PROGRAM demo3
VAR
	runner : FB_TaskRunner(ContainerType.PARALLEL_QUEUE);

	init: BOOL;
	_state :UINT;
	mc_power : FutureMCPower;
	_handl_power_on	: I_Job;
	_handl_demo_job : I_Job;
	
	_today : TIMESTRUCT;

	bPower : BOOL;
	bStart : BOOL;

	motion_data : ST_MotionData;	
	demo_job_container : FB_BatchJobContainer;
	i : UDINT;
END_VAR

IF NOT init THEN
	JobCreateDemo(demo_job_container, GVL.axis1); // demo_job にメソッドを通してシーケンスジョブを組み立てる
	mc_power.future_name := 'POWER_CTRL';
	init := TRUE;	// RUN 後 1 サイクルだけ実行
END_IF

_today := FILETIME64_TO_SYSTEMTIME(runner.current_time);
runner(root_job_name := 'ROOT',root_job_serial := (_today.wYear MOD 100) * 10000 + _today.wMonth * 100 + _today.wDay);

// Axis
GVL.axis1.ReadStatus();
MEMCPY(ADR(motion_data), ADR(GVL.axis1.NcToPlc), SIZEOF(GVL.axis1.NcToPlc));
motion_data.record_time := runner.current_time;

CASE _state OF
	0:
		IF bPower THEN
			mc_power.set_parameters(axis := GVL.axis1, status := TRUE); // Servo on
			_handl_power_on := runner.append_future(mc_power);
			_state := 1;
		END_IF
	1:
		IF _handl_power_on.ready THEN
			_handl_power_on.start();
		END_IF
		IF _handl_power_on.done THEN
			_state := 2;
		END_IF
	2:
		IF bStart THEN
			_handl_demo_job := runner.append_future(demo_job_container);
			_state := 3;
		END_IF
	3:
		IF _handl_demo_job.ready THEN
			_handl_demo_job.start();
		END_IF
		IF _handl_demo_job.current_state = E_FutureExecutionState.finish THEN
			_state := 2;
			//bStart := FALSE;
		END_IF
		IF NOT bPower THEN
			_state := 4;
		END_IF
	4:
		IF runner.halt(_handl_demo_job) THEN
			_state := 5;
		END_IF
	5:
		mc_power.set_parameters(axis := GVL.axis1, status := FALSE); // Servo off
		_handl_power_on := runner.append_future(mc_power);
		_state := 6;
	6:
		IF _handl_power_on.ready THEN
			_handl_power_on.start();
		END_IF
		IF _handl_power_on.done THEN
			_state := 0;
		END_IF
END_CASE

//IF _state > 0 AND NOT bPower THEN
//END_IF

METHOD JobCreateDemo : BOOL
VAR_INPUT
	job_container : I_Container;
	stAxis1	: REFERENCE TO AXIS_REF;
END_VAR
VAR
	_base_future : I_Future;
	_job_temp : I_Job;
	_job_temp_parent : I_Job;
	sleep : POINTER TO FutureSleep;
	sleep_creator : FutureSleepCreator;

	//mc_move_rel_future : POINTER TO FutureMCMoveRelative;
	mc_move_rel_future_creator : FutureMCMoveRelativeCreator;

	//mc_move_abs_future : POINTER TO FutureMCMoveAbsolute;
	mc_move_abs_future_creator : FutureMCMoveAbsoluteCreator;

	//mc_move_velocity_future: POINTER TO FutureMCMoveVelocity;
	mc_move_velocity_future_creator: FutureMCMoveVelocityCreator;
	
	mc_stop_future_creator : FutureMcStopCreator;
	
	i : UDINT;

END_VAR
//base_job.create_container(ContainerTYpe.BATCH, 'DEMO_JOB');
IF __QUERYINTERFACE(job_container,_base_future) THEN
	_base_future.future_name := 'JOB ROOT';
END_IF

// Sequence
_job_temp_parent := job_container.create_container(ContainerTYpe.BATCH, 'STEP MOVING');
FOR i := 1 TO 4 DO

	mc_move_rel_future_creator.set_parameters(stAxis1,20,200,0,0,0,0);
	_job_temp := _job_temp_parent.children.create_job(mc_move_rel_future_creator,'Move +20 deg, 200 deg/s');

	sleep_creator.sleep_time := T#100MS;
	_job_temp := _job_temp_parent.children.create_job(sleep_creator,'Wait 100ms');
	
END_FOR

// position set to 0

mc_move_abs_future_creator.set_parameters(stAxis1,0,200,0,0,0,0);
_job_temp := job_container.create_job(mc_move_abs_future_creator,'Back to home');

FOR i := 1 TO 10 DO

	mc_move_rel_future_creator.set_parameters(stAxis1,-20,200,0,0,0,0);
	_job_temp := job_container.create_job(mc_move_rel_future_creator,'Move -20 deg, 200 deg/s');

	sleep_creator.sleep_time := T#100MS;
	_job_temp := job_container.create_job(sleep_creator,'Wait 100ms');
	
END_FOR

// position to 0

mc_move_abs_future_creator.set_parameters(stAxis1,0,200,0,0,0,0);
_job_temp := job_container.create_job(mc_move_abs_future_creator,'Back to home');

sleep_creator.sleep_time := T#100MS;
_job_temp := job_container.create_job(sleep_creator,'Wait 100ms');

// 1000deg/s -> 500deg/s

mc_move_velocity_future_creator.set_parameters(stAxis1,MC_Direction.MC_Positive_Direction,10,0,0,0,0);
_job_temp := job_container.create_job(mc_move_velocity_future_creator,'Move velocity');

sleep_creator.sleep_time := T#5S;
_job_temp := job_container.create_job(sleep_creator,'10 deg/s 5 seconds');

mc_move_velocity_future_creator.set_parameters(stAxis1,MC_Direction.MC_Positive_Direction,100,0,0,0,0);
_job_temp := job_container.create_job(mc_move_velocity_future_creator,'Move velocity');

sleep_creator.sleep_time := T#5S;
_job_temp := job_container.create_job(sleep_creator,'100 deg/s 5 seconds');

mc_move_velocity_future_creator.set_parameters(stAxis1,MC_Direction.MC_Positive_Direction,250,0,0,0,0);
_job_temp := job_container.create_job(mc_move_velocity_future_creator,'Move velocity');

sleep_creator.sleep_time := T#5S;
_job_temp := job_container.create_job(sleep_creator,'250 deg/s 5 seconds');

mc_stop_future_creator.set_parameters(stAxis1,0,0);
_job_temp := job_container.create_job(mc_stop_future_creator,'STOP');

// position to 0

mc_move_abs_future_creator.set_parameters(stAxis1,0,250,0,0,0,0);
_job_temp := job_container.create_job(mc_move_abs_future_creator,'Back to home');
END_METHOD

END_PROGRAM

(* stored: Version 1.1.0.1, ProductVersion 3.1.4026.18
   POU demo3: Id {0711fc19-ddf5-4c28-b96d-7cde88b1723f}, SpecialFunc None
   Method JobCreateDemo: Id {c6c18e30-8bba-4c6d-806d-02b28dd2a277} *)
